# EPICS StreamDevice protocol: TektronixOscSup/tektronixOsc.proto
OutTerminator = '\n';
ReplyTimeout = 1000;

getIDN {
    out "*IDN?";
    #Read no more that 39 chars (EPICS limit)
    in "%/(.{0,39})/";
    ExtraInput = Ignore;
}

getYDATA {
    # Ask scope for y data points
    out ":VERBOSE 0;:HEADER 0;:DATA:SOURCE CH\$1;:DATA:START 1;:DATA:STOP 10000;:DATA:ENC ASCII;:DATA:WIDTH 1;:CURVE?";
    separator=",";
    in "%d";
    ExtraInput = Ignore;
}

getXINC {
    # Get x increment
    out ":DATA:SOURCE CH\$1;:WFMOUTPRE:XINCR?";
    in "%f";
    ExtraInput = Ignore;
}

getYMULT {
    # Get y multiplier
    out ":DATA:SOURCE CH\$1;:WFMOUTPRE:YMULT?";
    in "%f";
    ExtraInput = Ignore;
}

getXUNIT {
    # Get x unit
    out ":DATA:SOURCE CH\$1;:WFMOUTPRE:XUNIT?";
    in '%/([a-zA-Z]+)/';
    ExtraInput = Ignore;
}

getYUNIT {
    # Get y unit
    out ":DATA:SOURCE CH\$1;:WFMOUTPRE:YUNIT?";
    in '%/([a-zA-Z]+)/';
    ExtraInput = Ignore;
}

getXZERO {
    # Get the X start point (0)
    out ":DATA:SOURCE CH\$1;:WFMOUTPRE:XZERO?";
    in "%f";
    ExtraInput = Ignore;
}

getYZERO {
    # Get the Y start point (0)
    out ":DATA:SOURCE CH\$1;:WFMOUTPRE:YZERO?";
    in "%f";
    ExtraInput = Ignore;
}

getMeasurement {
    out "MEASU:MEAS\$1:VALUE?";
	in "%f";
    ExtraInput = Ignore;
	@init {
	    out "HEAD OFF";
	}
}
